PROGRAM pouEtherCATdiag
VAR
	iVal: WORD;
	tVal: WORD;
	tmask: WORD;
	state: UINT;
	i: UINT;
	decode:fb_decodeEtherCAT;
	
	retvall: UDINT;
	idbGetConfSlaves: FB_EcGetConfSlaves;
	test: BOOL;
	testams: BOOL;
	a: UINT;
	tDiagScreenSize: UINT;
	tDiagScreenWidth: UINT;
	tDiagScreenPointer: UINT;
	
	
	readcoe: FB_EcCoESdoRead;
	
	isCoeBusy: BOOL;
	isCoeError: BOOL;
	isCoecbRead: UDINT;
	currentReadNum: UINT;
	f: UINT;
END_VAR
VAR // added by the converter: edge detectors and wires of the graphical bodies
    _rt1, _rt2, _rt3 : R_TRIG;
END_VAR

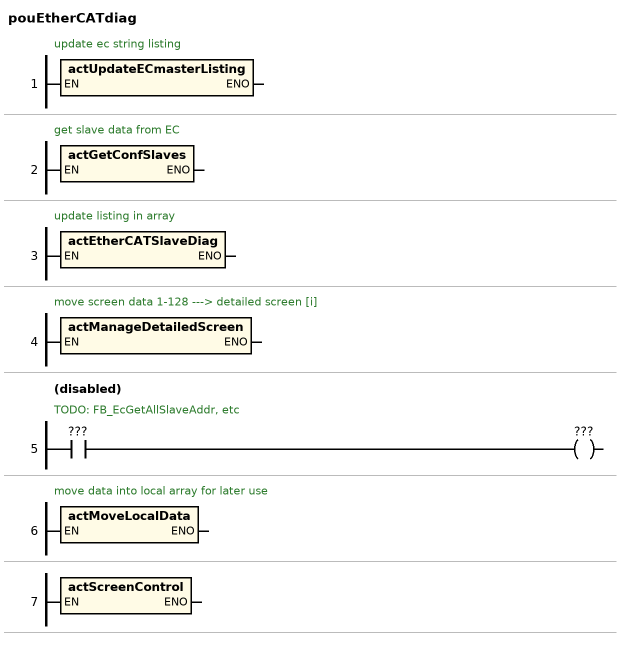
// NETWORK 1
// update ec string listing
actUpdateECmasterListing();

// NETWORK 2
// get slave data from EC
actGetConfSlaves();

// NETWORK 3
// update listing in array
actEtherCATSlaveDiag();

// NETWORK 4
// move screen data 1-128 ---> detailed screen [i]
actManageDetailedScreen();

// NETWORK 5 (disabled)
// TODO: FB_EcGetAllSlaveAddr, etc
// ??? := ???;

// NETWORK 6
// move data into local array for later use
actMoveLocalData();

// NETWORK 7
actScreenControl();

ACTION actEtherCATSlaveDiag:
IF System.PulseOneSecond THEN
	FOR i := 1 TO  etherCATdiag.maxNumEtherCATSlaves DO //
	
	////////////////////////////////////////////////////////////////
	//test write value
	//TODO: REMOVE
	//etherCATdiag.RawEtherCATStateDiag[i] := 16#8008; 
	//etherCATdiag.EtherCATslaveDiag[i].SlaveNumber := i;
	//etherCATdiag.EtherCATslaveDiag[i].crcCount.portA := i;
	/////////////////////////////////////////////////////////////////
	
	//move temp data from scan to temp declarations
	decode(iVal:=etherCATdiag.RawEtherCATStateDiag[i]);
	etherCATdiag.EtherCATslaveDiag[i].currentState.state := decode.state;
	etherCATdiag.EtherCATslaveDiag[i].currentState.suffix := decode.suffix;
	
		//check values for fault
		//current state
		IF etherCATdiag.EtherCATslaveDiag[i].currentState.state <> EtherCATstate.OP  OR //EtherCATstate.OP 
			etherCATdiag.EtherCATslaveDiag[i].currentState.suffix <> EtherCATSuffix.NoState THEN //EtherCATSuffix.NoState
			etherCATdiag.EtherCATslaveDiag[i].currentState.isFault := TRUE;
			ELSE
			etherCATdiag.EtherCATslaveDiag[i].currentState.isFault := FALSE;	
		END_IF
		
		//record outer box
		//record previous state, latching 
		IF etherCATdiag.EtherCATslaveDiag[i].currentState.isFault = FALSE AND 
		   etherCATdiag.EtherCATslaveDiag[i].historicalState.isFault = FALSE THEN
			//at this time, record the current state in the historical state
			etherCATdiag.EtherCATslaveDiag[i].historicalState.state := etherCATdiag.EtherCATslaveDiag[i].currentState.state;
			etherCATdiag.EtherCATslaveDiag[i].historicalState.suffix := etherCATdiag.EtherCATslaveDiag[i].currentState.suffix;
		END_IF
		
		//clear inner box when fault is resolved
		IF 	etherCATdiag.EtherCATslaveDiag[i].currentState.isFault = FALSE AND
		   gHMIButtons.btnReset THEN
		   etherCATdiag.EtherCATslaveDiag[i].historicalState.isFault := FALSE;
		END_IF
				//check if any suffix fault exits
				IF etherCATdiag.EtherCATslaveDiag[i].currentState.suffix > 1 THEN
					
					//check suffix
					CASE etherCATdiag.EtherCATslaveDiag[i].currentState.suffix OF 
					EtherCATSuffix.SlaveSignalsError					: 	etherCATdiag.EtherCATslaveDiag[i].currentState.colour := HMIColour.colourRed;
					EtherCATSuffix.InvalidVendor				: 	etherCATdiag.EtherCATslaveDiag[i].currentState.colour := HMIColour.colourRed;
					EtherCATSuffix.InitError 					: 	etherCATdiag.EtherCATslaveDiag[i].currentState.colour := HMIColour.colourRed;
					EtherCATSuffix.SlaveDisabled				:	etherCATdiag.EtherCATslaveDiag[i].currentState.colour := HMIColour.colourRed;
					EtherCATSuffix.SlaveNotPresent				: 	etherCATdiag.EtherCATslaveDiag[i].currentState.colour := HMIColour.colourRed;
					EtherCATSuffix.SlaveSignalsLinkError		:	etherCATdiag.EtherCATslaveDiag[i].currentState.colour := HMIColour.colourRed;
					EtherCATSuffix.SlaveSignalsMissingLink		:	etherCATdiag.EtherCATslaveDiag[i].currentState.colour := HMIColour.colourRed;
					EtherCATSuffix.SlaveSignalsUnExpectLink		:	etherCATdiag.EtherCATslaveDiag[i].currentState.colour := HMIColour.colourRed;
					EtherCATSuffix.CommsPortA					:	etherCATdiag.EtherCATslaveDiag[i].currentState.colour := HMIColour.colourRed;
					EtherCATSuffix.CommsPortB					:	etherCATdiag.EtherCATslaveDiag[i].currentState.colour := HMIColour.colourRed;
					EtherCATSuffix.CommsPortC					:	etherCATdiag.EtherCATslaveDiag[i].currentState.colour := HMIColour.colourRed;
					EtherCATSuffix.CommsPortD					:	etherCATdiag.EtherCATslaveDiag[i].currentState.colour := HMIColour.colourRed;
					END_CASE;
					
				ELSE
					//otherwise check state to get green
					CASE etherCATdiag.EtherCATslaveDiag[i].currentState.state OF 
					EtherCATstate.INIT		: 	etherCATdiag.EtherCATslaveDiag[i].currentState.colour := HMIColour.colourRed;
					EtherCATstate.PREOP		: 	etherCATdiag.EtherCATslaveDiag[i].currentState.colour := HMIColour.colourRed;
					EtherCATstate.BOOT		: 	etherCATdiag.EtherCATslaveDiag[i].currentState.colour := HMIColour.colourRed;
					EtherCATstate.SAFEOP	: 	etherCATdiag.EtherCATslaveDiag[i].currentState.colour := HMIColour.colourRed;
					EtherCATstate.OP		: 	etherCATdiag.EtherCATslaveDiag[i].currentState.colour := HMIColour.colourGreen;
					END_CASE;
					
				END_IF
	END_FOR
END_IF
END_ACTION

ACTION actGetCoEData:

//get slave id of each slave to read data from

//Index 1018 Identity

//data from beckhoff manuals
(*
1018:0 Identity Information for identifying the slave UINT8 RO 0x04 (4dec)
1018:01 Vendor ID Vendor ID of the EtherCAT slave UINT32 RO 0x00000002 (2dec)
1018:02 Product code Product code of the EtherCAT slave UINT32 RO 0x071B4052 (119226450dec)
1018:03 Revision Revision number of the EtherCAT slave; the Low Word (bit 0-15) indicates the special terminal number, the High Word (bit 16-31) refers to the  device description UINT32 RO 0x00000000 (0dec)
1018:04 Serial number Serial number of the EtherCAT slave; the Low Byte (bit 0-7) of the Low Word contains the year of production, the High Byte (bit 8-15) of the Low Word contains the week of production, the High Word (bit 16-31) is 0 UINT32 RO 0x00000000 (0dec) CoE parameters 162 Version: 3.7 EP1xxx
*)



//only input type modules?
(*
F900:02 Internal Temperature Internal temperature INT8 RO 0x00 (0dec)
F900:04 Voltage Us Measured value of the supply voltage US UINT16 RO 0x0000 (0dec)
*)



//only output type modules?
(*
F900:02 Internal Temperature INT8 RO 0x00 (0dec) 
F900:04 Voltage Us UINT16 RO 0x0000 (0dec)
F900:05 Voltage Up UINT16 RO 0x0000 (0dec)
*)

//zero counter
currentReadNum := 0;

//count out of scan for each entry of detected ethercat slave

//IF etherCATdiag.arryEcConfSlaveInfo[currentReadNum].


//read CoE data
readcoe(	sNetId:=,
			nSlaveAddr:=,
			nSubIndex:=,
			nIndex:=,
			pDstBuf:=,
			cbBufLen:=,
			bExecute:=,
			tTimeout:=T#5S
			);
			
isCoeBusy := readcoe.bBusy;
isCoeError := readcoe.bError;
isCoecbRead := readcoe.cbRead;
END_ACTION

ACTION actGetConfSlaves:
//convert AMSNETID type to string
idbGetConfSlaves.sNetId := F_CreateAmsNetId(nIds:=system.ecMasterData[1].ecAMSmaster);

//get slave info
idbGetConfSlaves(	sNetId 					:=,
					pArrEcConfSlaveInfo		:=ADR(etherCATdiag.arryEcConfSlaveInfo),
					cbBufLen				:=SIZEOF(etherCATdiag.arryEcConfSlaveInfo),
					bExecute				:=test,
					tTimeout				:=DEFAULT_ADS_TIMEOUT
				);
END_ACTION

ACTION actManageDetailedScreen:
//get max detail diag num
etherCATdiag.detailDiagNum	:= MAX(etherCATdiag.detailDiagNum, 1);

//move value from selected screen index (slave number) to the detail view
IF System.PulseOneSecond THEN
	retvall :=	MEMCPY( destAddr 		:=	ADR(etherCATdiag.detailDiag),
						srcAddr 		:=	ADR(etherCATdiag.diagScreen[etherCATdiag.detailDiagNum]),
						n 				:=	SIZEOF(etherCATdiag.detailDiag)
						);	
END_IF
END_ACTION

ACTION actMoveLocalData:
IF System.PulseOneSecond THEN
	//move data from FB_EcGetConfSlaves (etherCATdiag.arryEcConfSlaveInfo) to data for HMI
	FOR a := 1 TO etherCATdiag.maxNumEtherCATSlaves DO
		etherCATdiag.EtherCATslaveDiag[a].ConfigData := etherCATdiag.arryEcConfSlaveInfo[a];
	END_FOR
END_IF
END_ACTION

ACTION actScreenControl:
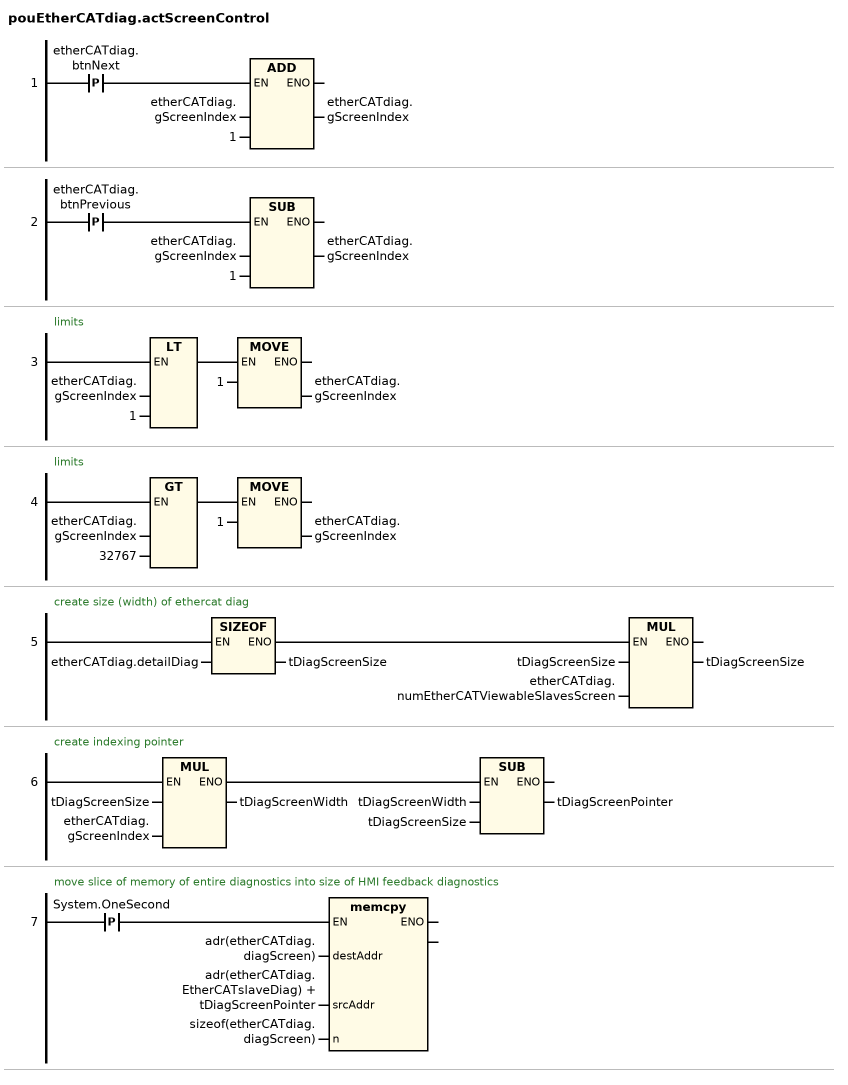
// NETWORK 1
_rt1(CLK := etherCATdiag.btnNext);
IF _rt1.Q THEN etherCATdiag.gScreenIndex := etherCATdiag.gScreenIndex + 1; END_IF

// NETWORK 2
_rt2(CLK := etherCATdiag.btnPrevious);
IF _rt2.Q THEN etherCATdiag.gScreenIndex := etherCATdiag.gScreenIndex - 1; END_IF

// NETWORK 3
// limits
IF etherCATdiag.gScreenIndex < 1 THEN etherCATdiag.gScreenIndex := 1; END_IF

// NETWORK 4
// limits
IF etherCATdiag.gScreenIndex > 32767 THEN etherCATdiag.gScreenIndex := 1; END_IF

// NETWORK 5
// create size (width) of ethercat diag
tDiagScreenSize := SIZEOF(etherCATdiag.detailDiag);
tDiagScreenSize := tDiagScreenSize * etherCATdiag.numEtherCATViewableSlavesScreen;

// NETWORK 6
// create indexing pointer
tDiagScreenWidth := tDiagScreenSize * etherCATdiag.gScreenIndex;
tDiagScreenPointer := tDiagScreenWidth - tDiagScreenSize;

// NETWORK 7
// move slice of memory of entire diagnostics into size of HMI feedback diagnostics
_rt3(CLK := System.OneSecond);
IF _rt3.Q THEN
    memcpy(destAddr := adr(etherCATdiag.diagScreen), srcAddr := adr(etherCATdiag.EtherCATslaveDiag) + tDiagScreenPointer, n := sizeof(etherCATdiag.diagScreen));
END_IF
END_ACTION

ACTION actUpdateECmasterListing:
//update array memory

IF System.PulseOneSecond THEN
	FOR f := 1 TO etherCATdiag.maxNumEtherCATmasters DO
		 IF system.ecMasterData[f].ecAMSmaster[0] > 1 THEN
			 //convert from byte to string for viewing
			 system.ecMasterData[f].ecAMSmasterstr := F_CreateAmsNetId(system.ecMasterData[f].ecAMSmaster);
			 
			 //move to internal memory
			 etherCATmasters.strActiveMastersList[f] := system.ecMasterData[f].ecAMSmasterstr;
		 END_IF
	END_FOR
END_IF
END_ACTION

END_PROGRAM

(* stored: Version 1.1.0.1, ProductVersion 3.1.4024.12
   POU pouEtherCATdiag: Id {73650198-8c30-49b6-b422-2b646bfaa17e}, SpecialFunc None
   Action actEtherCATSlaveDiag: Id {ad26e273-933b-4a92-8e3a-4cf2719bddff}
   Action actGetCoEData: Id {7fab3804-7adb-4c5b-bb8f-fc49082e9037}
   Action actGetConfSlaves: Id {0d22b66e-82b2-4403-abb6-b5b6d5ce9218}
   Action actManageDetailedScreen: Id {e0b81d8e-d637-494d-8072-e566ee9c1c33}
   Action actMoveLocalData: Id {07442dd0-a551-4aff-8d35-4ea4b270238f}
   Action actScreenControl: Id {4f5ebe78-f033-4000-933c-17c11db7a664}
   Action actUpdateECmasterListing: Id {8099666f-0b1c-4403-910b-3efdba95e88e} *)
